// TIA Portal V15.1 export
// export: Created 2024-06-21T08:40:53.758089Z, ExportSetting WithDefaults, DisplayName Totally Integrated Automation Portal, DisplayVersion V15.1 Update 5, DisplayName TIA Portal Openness, DisplayVersion V15.1 Update 5, DisplayName SINAMICS Startdrive Advanced, DisplayVersion V15.1, DisplayName G130, G150, S120, S150, SINAMICS MV, S210, DisplayVersion V15.1, DisplayName G110M, G120, G120C, G120D, G120P, DisplayVersion V15.1, DisplayName STEP 7 Professional, DisplayVersion V15.1 Update 5, DisplayName STEP 7 Safety, DisplayVersion V15.1, DisplayName WinCC Professional, DisplayVersion V15.1 Update 5, DisplayName SIMATIC Visualization Architect, DisplayVersion V15.1
FUNCTION "LHmiInterface" : Void   // FC1011, FBD
TITLE = LBitToWord
{ S7_Optimized_Access := 'FALSE' }
AUTHOR : VCC
FAMILY : Control
NAME : Bit2Word
VERSION : 1.0
// ================================================================================
// Moves the 16 input bits to one output word
// ================================================================================
// stored: AutoNumber false, IsIECCheckEnabled false, SetENOAutomatically False, UDAEnableTagReadback false
   VAR_INPUT
      I_0 : Bool;   // Input 0
      I_0_Txt : String;   // Input 0 - Description
      I_1 : Bool;   // Input 1
      I_1_Txt : String;   // Input 1 - Description
      I_2 : Bool;   // Input 2
      I_2_Txt : String;   // Input 2 - Description
      I_3 : Bool;   // Input 3
      I_3_Txt : String;   // Input 3 - Description
      I_4 : Bool;   // Input 4
      I_4_Txt : String;   // Input 4 - Description
      I_5 : Bool;   // Input 5
      I_5_Txt : String;   // Input 5 - Description
      I_6 : Bool;   // Input 6
      I_6_Txt : String;   // Input 6 - Description
      I_7 : Bool;   // Input 7
      I_7_Txt : String;   // Input 7 - Description
      I_8 : Bool;   // Input 8
      I_8_Txt : String;   // Input 8 - Description
      I_9 : Bool;   // Input 9
      I_9_Txt : String;   // Input 9 - Description
      I_10 : Bool;   // Input 10
      I_10_Txt : String;   // Input 10 - Description
      I_11 : Bool;   // Input 11
      I_11_Txt : String;   // Input 11 - Description
      I_12 : Bool;   // Input 12
      I_12_Txt : String;   // Input 12 - Description
      I_13 : Bool;   // Input 13
      I_13_Txt : String;   // Input 13 - Description
      I_14 : Bool;   // Input 14
      I_14_Txt : String;   // Input 14 - Description
      I_15 : Bool;   // Input 15
      I_15_Txt : String;   // Input 15 - Description
   END_VAR
   VAR_OUTPUT
      O_Word : Word;   // Output Word
      O_Txt : Struct   // Animation description of the bits
         "0" : String[50];   // Description
         "1" : String[50];   // Description
         "2" : String[50];   // Description
         "3" : String[50];   // Description
         "4" : String[50];   // Description
         "5" : String[50];   // Description
         "6" : String[50];   // Description
         "7" : String[50];   // Description
         "8" : String[50];   // Description
         "9" : String[50];   // Description
         "10" : String[50];   // Description
         "11" : String[50];   // Description
         "12" : String[50];   // Description
         "13" : String[50];   // Description
         "14" : String[50];   // Description
         "15" : String[50];   // Description
      END_STRUCT;
   END_VAR
BEGIN

REGION Network 1: **** 8 - Outputs ****
   // Move bit 0 to Word
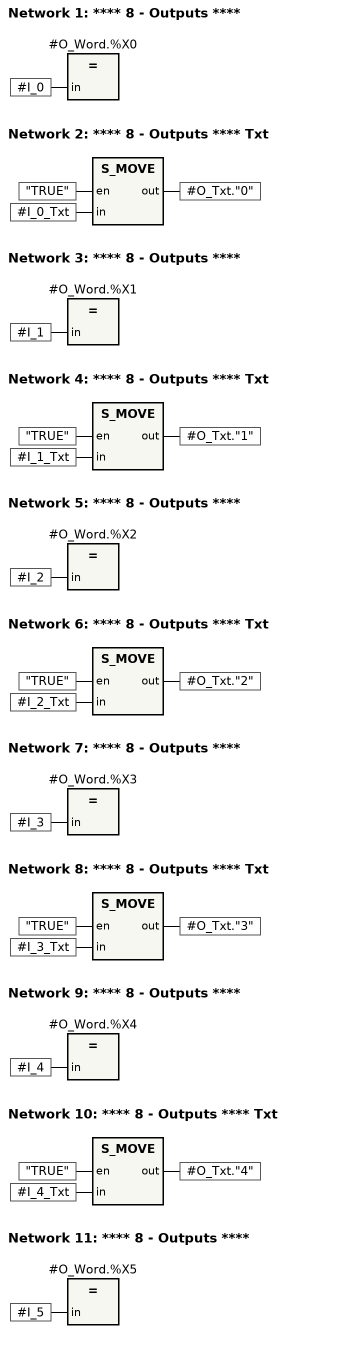
   #O_Word.%X0 := #I_0;
END_REGION

REGION Network 2: **** 8 - Outputs **** Txt
   IF "TRUE" THEN #O_Txt."0" := #I_0_Txt; END_IF;
END_REGION

REGION Network 3: **** 8 - Outputs ****
   // Move bit 1 to Word
   #O_Word.%X1 := #I_1;
END_REGION

REGION Network 4: **** 8 - Outputs **** Txt
   IF "TRUE" THEN #O_Txt."1" := #I_1_Txt; END_IF;
END_REGION

REGION Network 5: **** 8 - Outputs ****
   // Move bit 2 to Word
   #O_Word.%X2 := #I_2;
END_REGION

REGION Network 6: **** 8 - Outputs **** Txt
   IF "TRUE" THEN #O_Txt."2" := #I_2_Txt; END_IF;
END_REGION

REGION Network 7: **** 8 - Outputs ****
   // Move bit 3 to Word
   #O_Word.%X3 := #I_3;
END_REGION

REGION Network 8: **** 8 - Outputs **** Txt
   IF "TRUE" THEN #O_Txt."3" := #I_3_Txt; END_IF;
END_REGION

REGION Network 9: **** 8 - Outputs ****
   // Move bit 4 to Word
   #O_Word.%X4 := #I_4;
END_REGION

REGION Network 10: **** 8 - Outputs **** Txt
   IF "TRUE" THEN #O_Txt."4" := #I_4_Txt; END_IF;
END_REGION

REGION Network 11: **** 8 - Outputs ****
   // Move bit 5 to Word
   #O_Word.%X5 := #I_5;
END_REGION

REGION Network 12: **** 8 - Outputs **** Txt
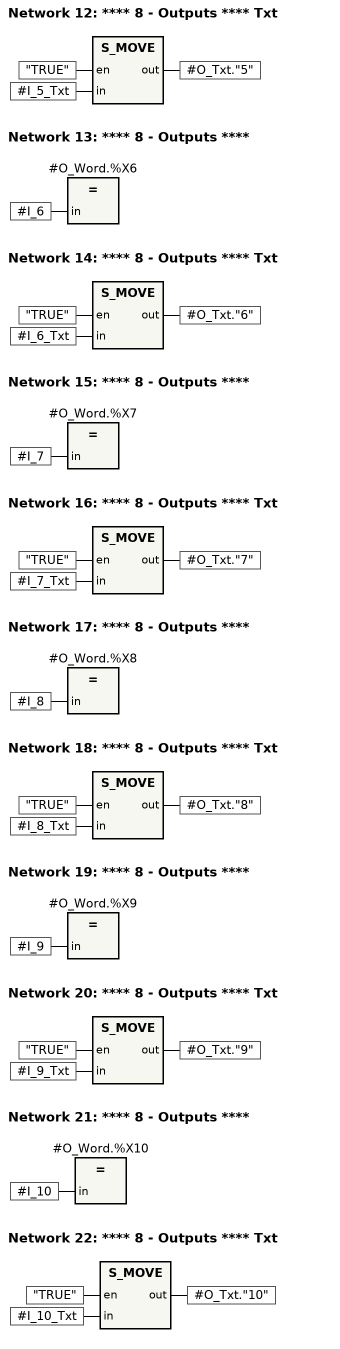
   IF "TRUE" THEN #O_Txt."5" := #I_5_Txt; END_IF;
END_REGION

REGION Network 13: **** 8 - Outputs ****
   // Move bit 6 to Word
   #O_Word.%X6 := #I_6;
END_REGION

REGION Network 14: **** 8 - Outputs **** Txt
   IF "TRUE" THEN #O_Txt."6" := #I_6_Txt; END_IF;
END_REGION

REGION Network 15: **** 8 - Outputs ****
   // Move bit 7 to Word
   #O_Word.%X7 := #I_7;
END_REGION

REGION Network 16: **** 8 - Outputs **** Txt
   IF "TRUE" THEN #O_Txt."7" := #I_7_Txt; END_IF;
END_REGION

REGION Network 17: **** 8 - Outputs ****
   // Move bit 8 to Word
   #O_Word.%X8 := #I_8;
END_REGION

REGION Network 18: **** 8 - Outputs **** Txt
   IF "TRUE" THEN #O_Txt."8" := #I_8_Txt; END_IF;
END_REGION

REGION Network 19: **** 8 - Outputs ****
   // Move bit 9 to Word
   #O_Word.%X9 := #I_9;
END_REGION

REGION Network 20: **** 8 - Outputs **** Txt
   IF "TRUE" THEN #O_Txt."9" := #I_9_Txt; END_IF;
END_REGION

REGION Network 21: **** 8 - Outputs ****
   // Move bit 10 to Word
   #O_Word.%X10 := #I_10;
END_REGION

REGION Network 22: **** 8 - Outputs **** Txt
   IF "TRUE" THEN #O_Txt."10" := #I_10_Txt; END_IF;
END_REGION

REGION Network 23: **** 8 - Outputs ****
   // Move bit 11 to Word
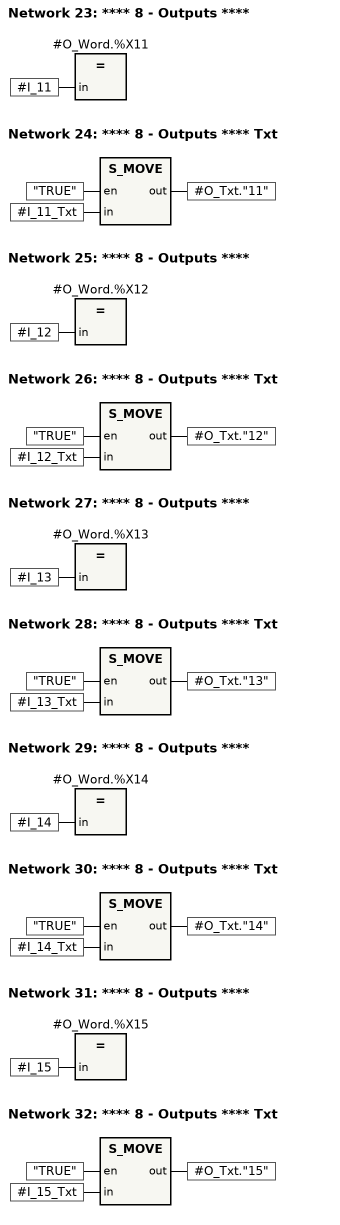
   #O_Word.%X11 := #I_11;
END_REGION

REGION Network 24: **** 8 - Outputs **** Txt
   IF "TRUE" THEN #O_Txt."11" := #I_11_Txt; END_IF;
END_REGION

REGION Network 25: **** 8 - Outputs ****
   // Move bit 12 to Word
   #O_Word.%X12 := #I_12;
END_REGION

REGION Network 26: **** 8 - Outputs **** Txt
   IF "TRUE" THEN #O_Txt."12" := #I_12_Txt; END_IF;
END_REGION

REGION Network 27: **** 8 - Outputs ****
   // Move bit 13 to Word
   #O_Word.%X13 := #I_13;
END_REGION

REGION Network 28: **** 8 - Outputs **** Txt
   IF "TRUE" THEN #O_Txt."13" := #I_13_Txt; END_IF;
END_REGION

REGION Network 29: **** 8 - Outputs ****
   // Move bit 14 to Word
   #O_Word.%X14 := #I_14;
END_REGION

REGION Network 30: **** 8 - Outputs **** Txt
   IF "TRUE" THEN #O_Txt."14" := #I_14_Txt; END_IF;
END_REGION

REGION Network 31: **** 8 - Outputs ****
   // Move bit 15 to Word
   #O_Word.%X15 := #I_15;
END_REGION

REGION Network 32: **** 8 - Outputs **** Txt
   IF "TRUE" THEN #O_Txt."15" := #I_15_Txt; END_IF;
END_REGION
END_FUNCTION
